PROGRAM MAIN
VAR
	nState : USINT := 0;

	fDividend : LREAL := 42.0; 
	fDivisor : LREAL := 1.0; // set to zero to force an error
	fQuotient : LREAL;
	
	// application POU using the result message interface to specify occurred errors (e.g. division by zero)
	fbMath : FB_MathCalculation := (eTraceLevel:=TcEventSeverity.Verbose); 
	
	// another application POU which encapsulates FB_MathCalculation
	fbCtrl : FB_Control := (eTraceLevel:=TcEventSeverity.Verbose); 
	
	sErrorText : STRING(255);
	bGetText : BOOL;
END_VAR

CASE nState OF
0: // calculation with fbMath
	fbMath.Division(fDividend:=fDividend, fDivisor:=fDivisor, fQuotient:=fQuotient);
	IF fbMath.bError THEN
		// error handling
		nState := 10;
	END_IF
	
1: // calculation with fbCtrl
	fbCtrl.Execute();
	IF fbCtrl.bError THEN
		// error handling
		// e.g. error text could be requested if execution failed.
		bGetText := TRUE;
		nState := 10;
	END_IF
	
10: // error occurred
	IF bGetText THEN
		IF fbCtrl.ipResultMessage.RequestEventText(	nLangId:=Tc3_EventLogger.GVL.nLangId_OnlineMonitoring, 
													sResult:=sErrorText, nResultSize:=SIZEOF(sErrorText) ) THEN
			bGetText := FALSE;
		END_IF
	END_IF
	
END_CASE

END_PROGRAM

(* stored: Version 1.1.0.1, ProductVersion 3.1.4022.10
   POU MAIN: Id {4e0d88d5-cdad-48a2-a95a-718032bb0b15}, SpecialFunc None *)
